(* PLC project top, Dassault Systèmes ControlBuild 2024x Refresh1 *)
(* stored: creationDateTime 2024-03-14T15:54:11-01:00 *)

PROGRAM a1

(* FBD diagram, written out as Structured Text *)
END_PROGRAM

PROGRAM a2

(* FBD diagram, written out as Structured Text *)
END_PROGRAM

PROGRAM sub_pou

(* FBD diagram, written out as Structured Text *)
END_PROGRAM

PROGRAM a3

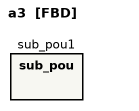
(* FBD diagram, written out as Structured Text *)
sub_pou1();
END_PROGRAM

PROGRAM my_app.top

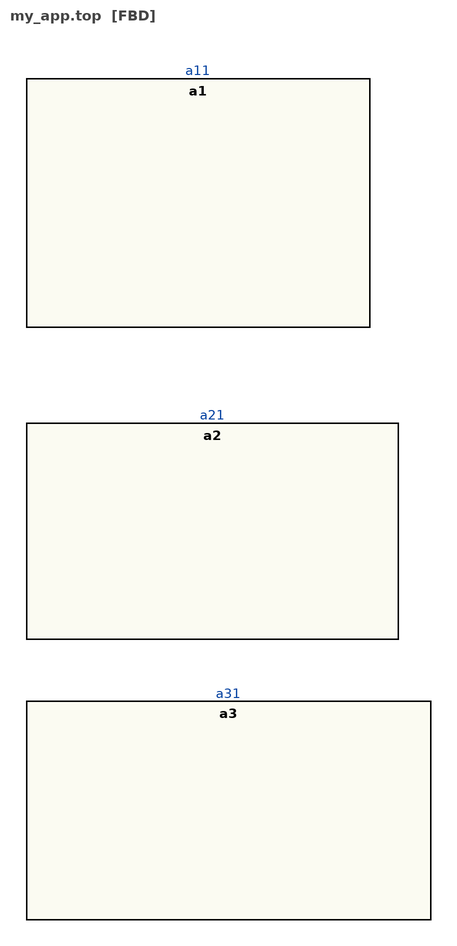
(* FBD diagram, written out as Structured Text *)
a11();
a21();
a31();
END_PROGRAM
